PROGRAM PRG_TcpTest
VAR
	fbTcp    : FB_MbTransportTcp := (sHost := '127.0.0.1', nPort := 502);
	fbDev    : FB_Mb_TestGood;
	stLog    : ST_MbLog;
	bTcpPass : BOOL;
END_VAR

fbTcp();
fbDev(itfTransport := fbTcp, nUnitId := 1, bEnable := TRUE, refLog := stLog);

bTcpPass := fbTcp.bConnected AND fbDev.bOnline
            AND (fbDev.Hr1.fValue = 1234) AND (fbDev.Hr2.fValue = 50.0) AND (fbDev.Hr3.fValue = 1.5);

END_PROGRAM

(* stored: Version 1.1.0.1
   POU PRG_TcpTest: Id {ca6b4fd9-bcce-4fa2-97ca-7295a7787863}, SpecialFunc None *)
